// TIA Portal V18 export
// export: Created 2026-03-12T16:04:35.0974227Z, ExportSetting WithDefaults, DisplayName Totally Integrated Automation Portal, DisplayVersion V18 Update 5, DisplayName TIA Portal Openness, DisplayVersion V18 Update 5, DisplayName TIA Portal Version Control Interface, DisplayVersion V18, DisplayName SINAMICS Startdrive Advanced, DisplayVersion V18, DisplayName SINAMICS Startdrive G130, G150, S120, S150, SINAMICS MV, S210, DisplayVersion V18, DisplayName SINAMICS Startdrive G110M, G120, G120C, G120D, G120P, G115D, DisplayVersion V18, DisplayName STEP 7 Professional, DisplayVersion V18 Update 5, DisplayName STEP 7 Safety, DisplayVersion V18, DisplayName WinCC Professional, DisplayVersion V18 Update 5
FUNCTION_BLOCK "FB FALHA"   // FB9, LAD
TITLE = Function Block FALHA - Falha dos motores/bombas
{ S7_Optimized_Access := 'TRUE' }
VERSION : 0.1
// Network 1: Condição SET-RESET da Falha da bomba
// stored: AutoNumber true, IsIECCheckEnabled false, IsRetainMemResEnabled false, MemoryReserve 100, SetENOAutomatically false, UDAEnableTagReadback false
   VAR_INPUT
      INPUT_FALHA : Bool;   // Entrada do sinal de falha instanciado na Network 1
      INPUT_TEMPO_RESET : Time;   // Tempo em segundos que a bomba irá resetar após identificar sem falha
      INPUT_TEMPO_NÃO_LIGOU : Time;   // Se após ligar a bomba não retornar o sinal de LIGADO pelo tempo configurado, aciona falha
      INPUT_LIGADO : Bool;   // Entrada do sinal de Motor/Bomba ligado
      INPUT_RESET_FALHA : Bool;   // Resetar a falha manualmente caso o sinal de INPUT_FALHA esteja FALSE
      INPUT_SAIDA_LIGA_BOMBA : Bool;   // Saída para ligar a bomba acionada
      INPUT_HABILITA_CONJUNTO : Bool;   // Identificação do conjunto de bombas (principal e reserva)
      INPUT_MANUTENCAO : Bool;   // Entrada responsavel por mudar o estado do equipamento em manut, sendo sem falha ativa.
   END_VAR
   VAR_OUTPUT
      FALHA : Bool;   // Saída do sinal de falha da instância do FB para o FC
      RESET_FALHA_INVERSOR : Bool;   // Reset sinal de falha do inversor de frequência
      FALHA_NÃO_LIGOU : Bool;
   END_VAR
   VAR
      NÃO_LIGOU : Bool;   // Sinal indicando que a bomba não ligou após comando, entrando em falha
      SET_FALHA : Bool;   // Memória auxiliar para o recebimento da falha
      TIMER_1 : IEC_TIMER;   // Temporizador para resetar a Falha
      TIMER_2 : IEC_TIMER;   // Temporizador para entrar em Falha
      LIGA_BOMBA_AUX { S7_SetPoint := 'True'} : Bool;   // Memória auxiliar para disparo do final de falha
   END_VAR
   VAR_TEMP   // added for the SCL form of the ladder/FBD networks
      _w1 : Bool;
   END_VAR
BEGIN

REGION Network 1: Saída do sinal de falha da instância do FB para o FC
   // Tratamento de falha da bomba
   // INPUT_FALHA: Entrada do sinal de falha instanciado na Network 1.
   // INPUT_TEMPO_RESET: Tempo em segundos que a bomba irá resetar após identificar sem falha.
   // INPUT_TEMPO_NÃO_LIGOU: Se após ligar a bomba não retornar o sinal de LIGADO pelo tempo configurado, aciona falha.
   // INPUT_LIGADO: Entrada do sinal de Motor/Bomba ligado
   // INPUT_RESET_FALHA: Resetar a falha manualmente caso o sinal de INPUT_FALHA esteja FALSE
   // NÃO_LIGOU: Memória auxiliar para acionar falha caso a bomba não retorno seu status de ligada.
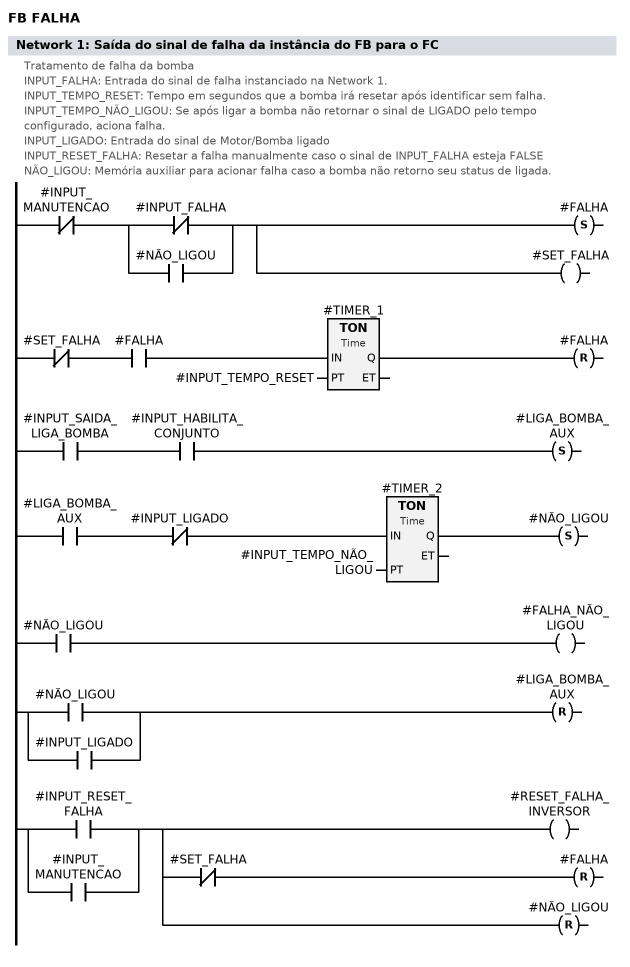
   RUNG wire#powerrail
      I_Contact( #INPUT_MANUTENCAO )
      wire#w1
      I_Contact( #INPUT_FALHA )
      wire#w2
      S_Coil( #FALHA )
   END_RUNG
   RUNG wire#w1
      Contact( #NÃO_LIGOU )
   END_RUNG wire#w2
   RUNG wire#w2
      Coil( #SET_FALHA )
   END_RUNG
   RUNG wire#powerrail
      I_Contact( #SET_FALHA )
      Contact( #FALHA )
      { S7_Templates := "time_type := Time" } #TIMER_1.TON(pt := #INPUT_TEMPO_RESET, et =>)
      R_Coil( #FALHA )
   END_RUNG
   RUNG wire#powerrail
      Contact( #INPUT_SAIDA_LIGA_BOMBA )
      Contact( #INPUT_HABILITA_CONJUNTO )
      S_Coil( #LIGA_BOMBA_AUX )
   END_RUNG
   RUNG wire#powerrail
      Contact( #LIGA_BOMBA_AUX )
      I_Contact( #INPUT_LIGADO )
      { S7_Templates := "time_type := Time" } #TIMER_2.TON(pt := #INPUT_TEMPO_NÃO_LIGOU, et =>)
      S_Coil( #NÃO_LIGOU )
   END_RUNG
   RUNG wire#powerrail
      Contact( #NÃO_LIGOU )
      Coil( #FALHA_NÃO_LIGOU )
   END_RUNG
   RUNG wire#powerrail
      Contact( #NÃO_LIGOU )
      wire#w3
      R_Coil( #LIGA_BOMBA_AUX )
   END_RUNG
   RUNG wire#powerrail
      Contact( #INPUT_LIGADO )
   END_RUNG wire#w3
   RUNG wire#powerrail
      Contact( #INPUT_RESET_FALHA )
      wire#w4
      Coil( #RESET_FALHA_INVERSOR )
   END_RUNG
   RUNG wire#powerrail
      Contact( #INPUT_MANUTENCAO )
   END_RUNG wire#w4
   RUNG wire#w4
      I_Contact( #SET_FALHA )
      R_Coil( #FALHA )
   END_RUNG
   RUNG wire#w4
      R_Coil( #NÃO_LIGOU )
   END_RUNG
   // the same network as SCL:
   #_w1 := NOT #INPUT_MANUTENCAO AND (NOT #INPUT_FALHA OR #NÃO_LIGOU);
   IF #_w1 THEN #FALHA := TRUE; END_IF;
   #SET_FALHA := #_w1;
   #TIMER_1.TON(IN := NOT #SET_FALHA AND #FALHA, PT := #INPUT_TEMPO_RESET);
   IF #TIMER_1.Q THEN #FALHA := FALSE; END_IF;
   IF #INPUT_SAIDA_LIGA_BOMBA AND #INPUT_HABILITA_CONJUNTO THEN #LIGA_BOMBA_AUX := TRUE; END_IF;
   #TIMER_2.TON(IN := #LIGA_BOMBA_AUX AND NOT #INPUT_LIGADO, PT := #INPUT_TEMPO_NÃO_LIGOU);
   IF #TIMER_2.Q THEN #NÃO_LIGOU := TRUE; END_IF;
   #FALHA_NÃO_LIGOU := #NÃO_LIGOU;
   IF #NÃO_LIGOU OR #INPUT_LIGADO THEN #LIGA_BOMBA_AUX := FALSE; END_IF;
   #RESET_FALHA_INVERSOR := #INPUT_RESET_FALHA OR #INPUT_MANUTENCAO;
   IF #RESET_FALHA_INVERSOR AND NOT #SET_FALHA THEN #FALHA := FALSE; END_IF;
   IF #RESET_FALHA_INVERSOR THEN #NÃO_LIGOU := FALSE; END_IF;
END_REGION
END_FUNCTION_BLOCK
